{attribute addProperty BoxType "EL2032--0000"}
{attribute addProperty Id "DiagAT %I*ARRAY[0..1] OF Diag_4CD4E3A21620ChannelAT %Q*ARRAY[0..1] OF Channel_7F374EB01620WcStateAT %I*WcState_F855686C1620InfoDataAT %I*InfoData_192954DE1620"}
{attribute addProperty CRC "1711085282"}
{attribute addProperty SizeInBites "64"}
{attribute addProperty SizeInBytes "8"}
TYPE EL2032_1D732299 :
STRUCT
	{attribute addProperty Name "Diag"}
	Diag : ARRAY[0..1] OF Diag_4CD4E3A2;
	{attribute addProperty Name "Channel"}
	Channel : ARRAY[0..1] OF Channel_7F374EB0;
	{attribute addProperty Name "WcState"}
	WcState : WcState_F855686C;
	{attribute addProperty Name "InfoData"}
	InfoData : InfoData_192954DE;
END_STRUCT
END_TYPE

(* stored: Version 1.2.0.0, ProductVersion 3.1.4024.9
   DUT EL2032_1D732299: Id {9b20023f-be2a-49ab-af4c-70467d097340} *)
